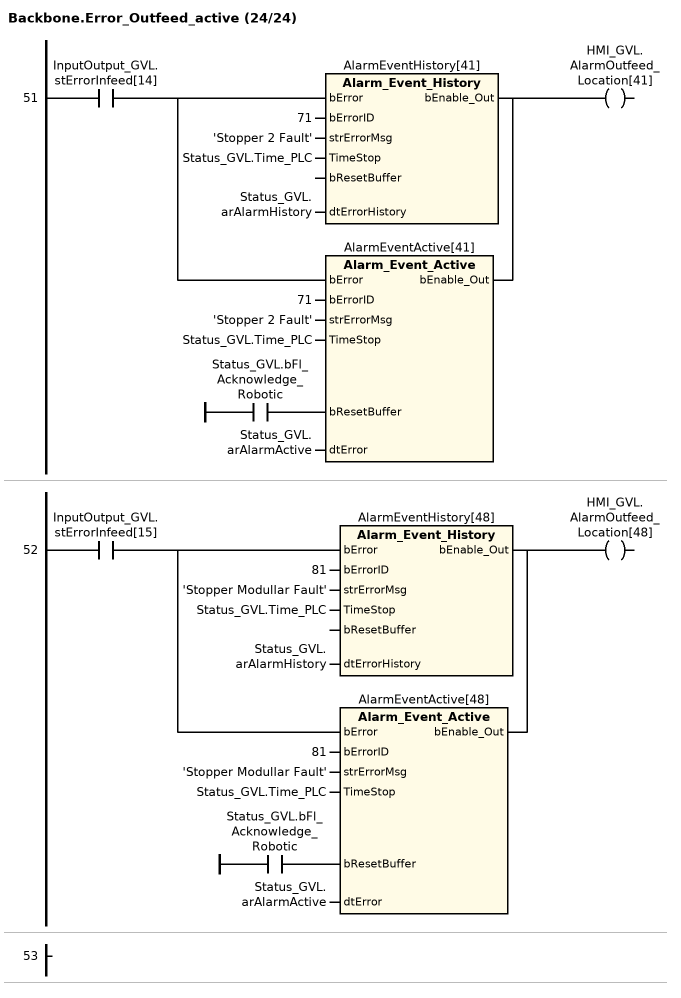
// NETWORK 51
AlarmEventHistory[41](
    bError := InputOutput_GVL.stErrorInfeed[14],
    bErrorID := 71,
    strErrorMsg := 'Stopper 2 Fault',
    TimeStop := Status_GVL.Time_PLC,
    dtErrorHistory := Status_GVL.arAlarmHistory); // Alarm_Event_History
AlarmEventActive[41](
    bError := InputOutput_GVL.stErrorInfeed[14],
    bErrorID := 71,
    strErrorMsg := 'Stopper 2 Fault',
    TimeStop := Status_GVL.Time_PLC,
    bResetBuffer := Status_GVL.bFl_Acknowledge_Robotic,
    dtError := Status_GVL.arAlarmActive); // Alarm_Event_Active
HMI_GVL.AlarmOutfeed_Location[41] := AlarmEventHistory[41].bEnable_Out OR AlarmEventActive[41].bEnable_Out;

// NETWORK 52
AlarmEventHistory[48](
    bError := InputOutput_GVL.stErrorInfeed[15],
    bErrorID := 81,
    strErrorMsg := 'Stopper Modullar Fault',
    TimeStop := Status_GVL.Time_PLC,
    dtErrorHistory := Status_GVL.arAlarmHistory); // Alarm_Event_History
AlarmEventActive[48](
    bError := InputOutput_GVL.stErrorInfeed[15],
    bErrorID := 81,
    strErrorMsg := 'Stopper Modullar Fault',
    TimeStop := Status_GVL.Time_PLC,
    bResetBuffer := Status_GVL.bFl_Acknowledge_Robotic,
    dtError := Status_GVL.arAlarmActive); // Alarm_Event_Active
HMI_GVL.AlarmOutfeed_Location[48] := AlarmEventHistory[48].bEnable_Out OR AlarmEventActive[48].bEnable_Out;

// NETWORK 53
END_ACTION

ACTION FGHS_DataCollect_active:
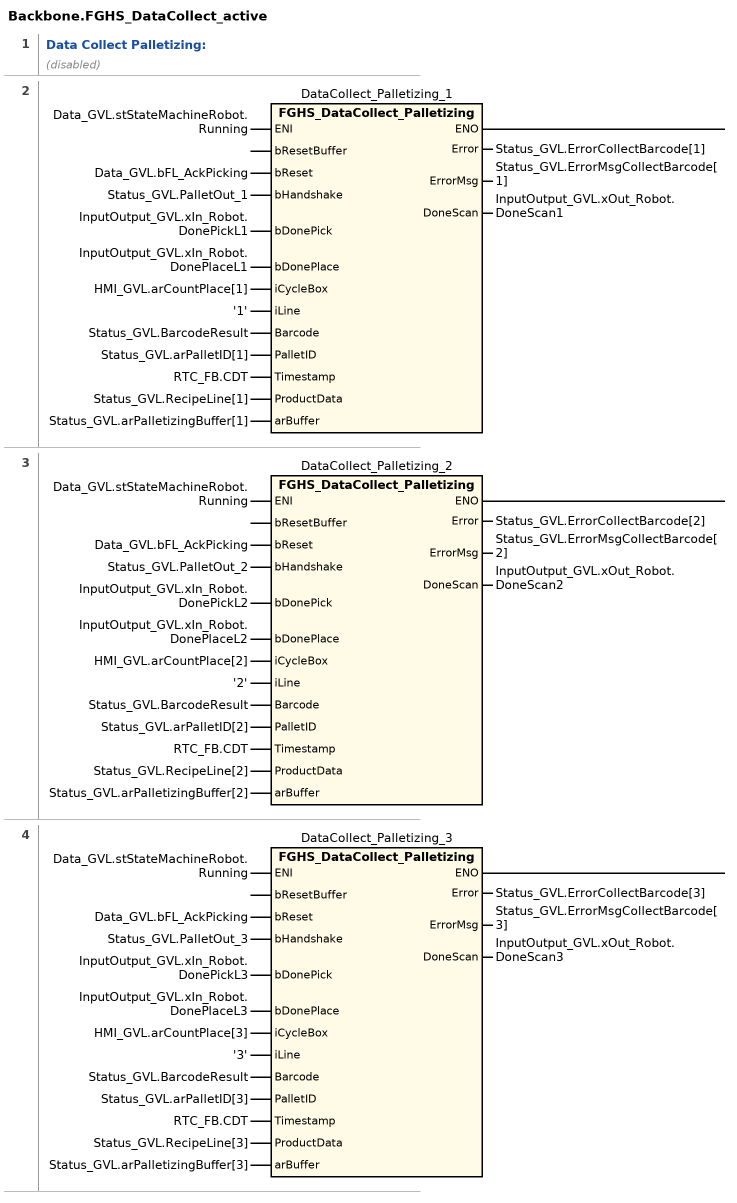
// NETWORK 1 (disabled)
// label: Data Collect Palletizing

// NETWORK 2
DataCollect_Palletizing_1(
    ENI := Data_GVL.stStateMachineRobot.Running,
    bReset := Data_GVL.bFL_AckPicking,
    bHandshake := Status_GVL.PalletOut_1,
    bDonePick := InputOutput_GVL.xIn_Robot.DonePickL1,
    bDonePlace := InputOutput_GVL.xIn_Robot.DonePlaceL1,
    iCycleBox := HMI_GVL.arCountPlace[1],
    iLine := '1',
    Barcode := Status_GVL.BarcodeResult,
    PalletID := Status_GVL.arPalletID[1],
    Timestamp := RTC_FB.CDT,
    ProductData := Status_GVL.RecipeLine[1],
    arBuffer := Status_GVL.arPalletizingBuffer[1],
    Error => Status_GVL.ErrorCollectBarcode[1],
    ErrorMsg => Status_GVL.ErrorMsgCollectBarcode[1],
    DoneScan => InputOutput_GVL.xOut_Robot.DoneScan1); // FGHS_DataCollect_Palletizing

// NETWORK 3
DataCollect_Palletizing_2(
    ENI := Data_GVL.stStateMachineRobot.Running,
    bReset := Data_GVL.bFL_AckPicking,
    bHandshake := Status_GVL.PalletOut_2,
    bDonePick := InputOutput_GVL.xIn_Robot.DonePickL2,
    bDonePlace := InputOutput_GVL.xIn_Robot.DonePlaceL2,
    iCycleBox := HMI_GVL.arCountPlace[2],
    iLine := '2',
    Barcode := Status_GVL.BarcodeResult,
    PalletID := Status_GVL.arPalletID[2],
    Timestamp := RTC_FB.CDT,
    ProductData := Status_GVL.RecipeLine[2],
    arBuffer := Status_GVL.arPalletizingBuffer[2],
    Error => Status_GVL.ErrorCollectBarcode[2],
    ErrorMsg => Status_GVL.ErrorMsgCollectBarcode[2],
    DoneScan => InputOutput_GVL.xOut_Robot.DoneScan2); // FGHS_DataCollect_Palletizing

// NETWORK 4
DataCollect_Palletizing_3(
    ENI := Data_GVL.stStateMachineRobot.Running,
    bReset := Data_GVL.bFL_AckPicking,
    bHandshake := Status_GVL.PalletOut_3,
    bDonePick := InputOutput_GVL.xIn_Robot.DonePickL3,
    bDonePlace := InputOutput_GVL.xIn_Robot.DonePlaceL3,
    iCycleBox := HMI_GVL.arCountPlace[3],
    iLine := '3',
    Barcode := Status_GVL.BarcodeResult,
    PalletID := Status_GVL.arPalletID[3],
    Timestamp := RTC_FB.CDT,
    ProductData := Status_GVL.RecipeLine[3],
    arBuffer := Status_GVL.arPalletizingBuffer[3],
    Error => Status_GVL.ErrorCollectBarcode[3],
    ErrorMsg => Status_GVL.ErrorMsgCollectBarcode[3],
    DoneScan => InputOutput_GVL.xOut_Robot.DoneScan3); // FGHS_DataCollect_Palletizing

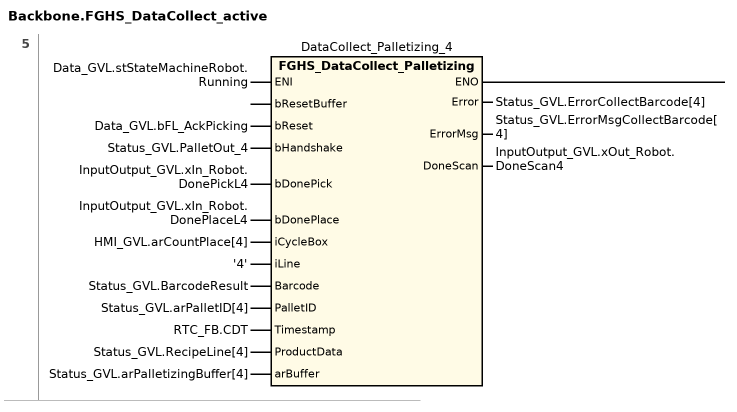
// NETWORK 5
DataCollect_Palletizing_4(
    ENI := Data_GVL.stStateMachineRobot.Running,
    bReset := Data_GVL.bFL_AckPicking,
    bHandshake := Status_GVL.PalletOut_4,
    bDonePick := InputOutput_GVL.xIn_Robot.DonePickL4,
    bDonePlace := InputOutput_GVL.xIn_Robot.DonePlaceL4,
    iCycleBox := HMI_GVL.arCountPlace[4],
    iLine := '4',
    Barcode := Status_GVL.BarcodeResult,
    PalletID := Status_GVL.arPalletID[4],
    Timestamp := RTC_FB.CDT,
    ProductData := Status_GVL.RecipeLine[4],
    arBuffer := Status_GVL.arPalletizingBuffer[4],
    Error => Status_GVL.ErrorCollectBarcode[4],
    ErrorMsg => Status_GVL.ErrorMsgCollectBarcode[4],
    DoneScan => InputOutput_GVL.xOut_Robot.DoneScan4); // FGHS_DataCollect_Palletizing
END_ACTION

ACTION FGHS_DataTraffict_active:
(* ============= Barcode Product ================= *)
//Line 1
	IF HMI_GVL.arCountReal[1] <> CheckCounter[1] THEN
		FOR Index[1] := 1 TO 60 BY 1 DO
		Status_GVL.arBarcodePallet[1,Index[1]]			:= Status_GVL.arPalletizingBuffer[1].BarcodeProduct[Index[1]];
		Status_GVL.arBarcodePalletTime[1,Index[1]]		:= Status_GVL.arPalletizingBuffer[1].BarcodeProductTime[Index[1]];
		Status_GVL.arDataPallet1[Index[1]].BarcodePallet	:= Status_GVL.arBarcodePallet[1,Index[1]];
		Status_GVL.arDataPallet1[Index[1]].BarcodePalletTime:= Status_GVL.arBarcodePalletTime[1,Index[1]]; 
		END_FOR
		CheckCounter[1]	:= HMI_GVL.arCountReal[1];
	END_IF
	
//Line 2
	IF HMI_GVL.arCountReal[2] <> CheckCounter[2] THEN
		FOR Index[2] := 1 TO 60 BY 1 DO
		Status_GVL.arBarcodePallet[2,Index[2]]			:= Status_GVL.arPalletizingBuffer[2].BarcodeProduct[Index[2]];
		Status_GVL.arBarcodePalletTime[2,Index[2]]		:= Status_GVL.arPalletizingBuffer[2].BarcodeProductTime[Index[2]];
		Status_GVL.arDataPallet2[Index[2]].BarcodePallet	:= Status_GVL.arBarcodePallet[2,Index[2]];
		Status_GVL.arDataPallet2[Index[2]].BarcodePalletTime:= Status_GVL.arBarcodePalletTime[2,Index[2]]; 
		END_FOR
		CheckCounter[2]	:= HMI_GVL.arCountReal[2];
	END_IF
	
//Line 3
	IF HMI_GVL.arCountReal[3] <> CheckCounter[3] THEN
		FOR Index[3] := 1 TO 60 BY 1 DO
		Status_GVL.arBarcodePallet[3,Index[3]]			:= Status_GVL.arPalletizingBuffer[3].BarcodeProduct[Index[3]];
		Status_GVL.arBarcodePalletTime[3,Index[3]]		:= Status_GVL.arPalletizingBuffer[3].BarcodeProductTime[Index[3]];
		Status_GVL.arDataPallet3[Index[3]].BarcodePallet	:= Status_GVL.arBarcodePallet[3,Index[3]];
		Status_GVL.arDataPallet3[Index[3]].BarcodePalletTime:= Status_GVL.arBarcodePalletTime[3,Index[3]]; 
		END_FOR
		CheckCounter[3]	:= HMI_GVL.arCountReal[3];
	END_IF
	
//Line 4
	IF HMI_GVL.arCountReal[4] <> CheckCounter[4] THEN
		FOR Index[4] := 1 TO 60 BY 1 DO
		Status_GVL.arBarcodePallet[4,Index[4]]			:= Status_GVL.arPalletizingBuffer[4].BarcodeProduct[Index[4]];
		Status_GVL.arBarcodePalletTime[4,Index[4]]		:= Status_GVL.arPalletizingBuffer[4].BarcodeProductTime[Index[4]];
		Status_GVL.arDataPallet4[Index[4]].BarcodePallet	:= Status_GVL.arBarcodePallet[4,Index[4]];
		Status_GVL.arDataPallet4[Index[4]].BarcodePalletTime:= Status_GVL.arBarcodePalletTime[4,Index[4]]; 
		END_FOR
		CheckCounter[4]	:= HMI_GVL.arCountReal[4];
	END_IF
	
	
(* ============= Link Up ================= *)
Status_GVl.arPallet_LinkUp[1]	:= Status_GVL.RecipeLine[1].LinkUpSource;
Status_GVl.arPallet_LinkUp[2]	:= Status_GVL.RecipeLine[2].LinkUpSource;
Status_GVl.arPallet_LinkUp[3]	:= Status_GVL.RecipeLine[3].LinkUpSource;
Status_GVl.arPallet_LinkUp[4]	:= Status_GVL.RecipeLine[4].LinkUpSource;


(* ============= EAN Variant ================= *)
Status_GVL.arCurrent_EAN[1]		:= Status_GVL.RecipeLine[1].EANVariant;
Status_GVL.arCurrent_EAN[2]		:= Status_GVL.RecipeLine[2].EANVariant;
Status_GVL.arCurrent_EAN[3]		:= Status_GVL.RecipeLine[3].EANVariant;
Status_GVL.arCurrent_EAN[4]		:= Status_GVL.RecipeLine[4].EANVariant;

(* ============= Code Variant ================= *)
Status_GVL.arCurrent_CodeVariant[1]		:= Status_GVL.RecipeLine[1].CodeVariant;
Status_GVL.arCurrent_CodeVariant[2]		:= Status_GVL.RecipeLine[2].CodeVariant;
Status_GVL.arCurrent_CodeVariant[3]		:= Status_GVL.RecipeLine[3].CodeVariant;
Status_GVL.arCurrent_CodeVariant[4]		:= Status_GVL.RecipeLine[4].CodeVariant;

(* ============= Interlock Infeed ================= *)
Status_GVL.ModullarInfeedBusy	:= InputOutput_GVL.Digital_Output[45];
END_ACTION

ACTION Indicator_active:
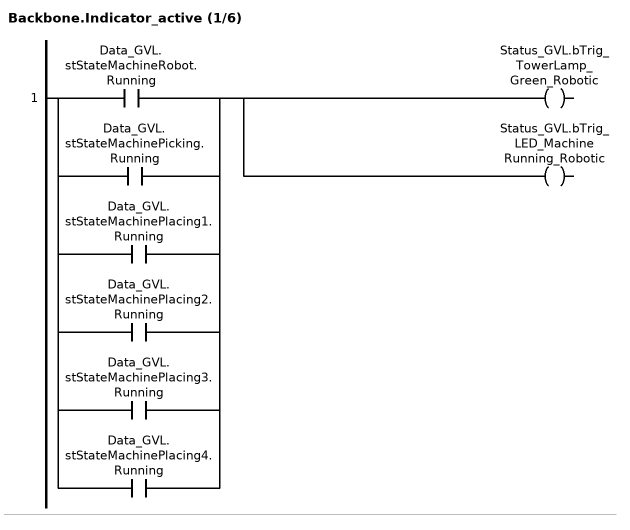
// NETWORK 1
_w1 := Data_GVL.stStateMachineRobot.Running OR Data_GVL.stStateMachinePicking.Running OR Data_GVL.stStateMachinePlacing1.Running OR Data_GVL.stStateMachinePlacing2.Running OR Data_GVL.stStateMachinePlacing3.Running OR Data_GVL.stStateMachinePlacing4.Running;
Status_GVL.bTrig_TowerLamp_Green_Robotic := _w1;
Status_GVL.bTrig_LED_MachineRunning_Robotic := _w1;

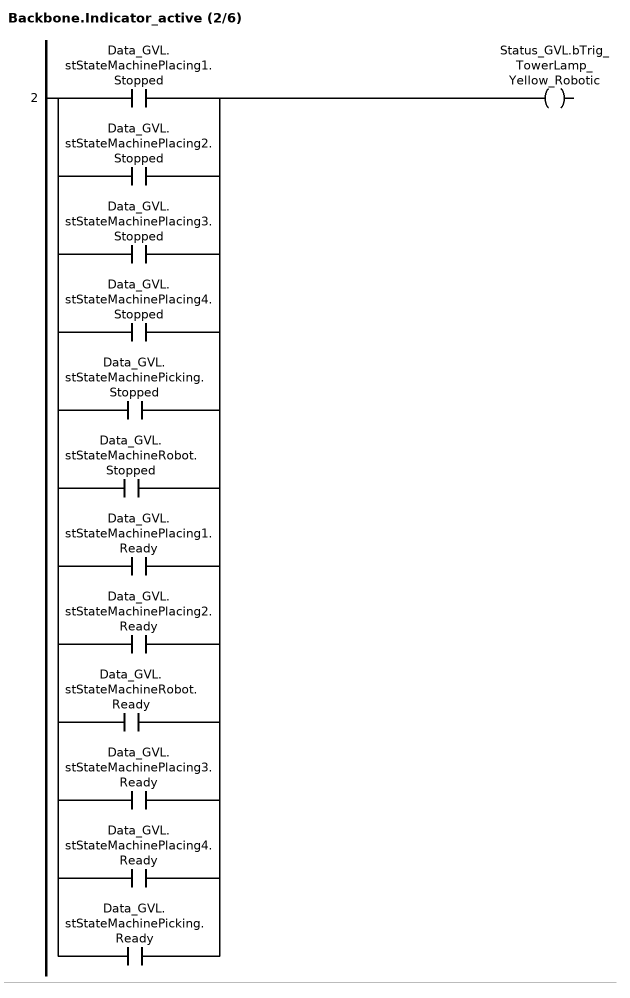
// NETWORK 2
Status_GVL.bTrig_TowerLamp_Yellow_Robotic := Data_GVL.stStateMachinePlacing1.Stopped OR Data_GVL.stStateMachinePlacing2.Stopped OR Data_GVL.stStateMachinePlacing3.Stopped OR Data_GVL.stStateMachinePlacing4.Stopped OR Data_GVL.stStateMachinePicking.Stopped OR Data_GVL.stStateMachineRobot.Stopped OR Data_GVL.stStateMachinePlacing1.Ready OR Data_GVL.stStateMachinePlacing2.Ready OR Data_GVL.stStateMachineRobot.Ready OR Data_GVL.stStateMachinePlacing3.Ready OR Data_GVL.stStateMachinePlacing4.Ready OR Data_GVL.stStateMachinePicking.Ready;

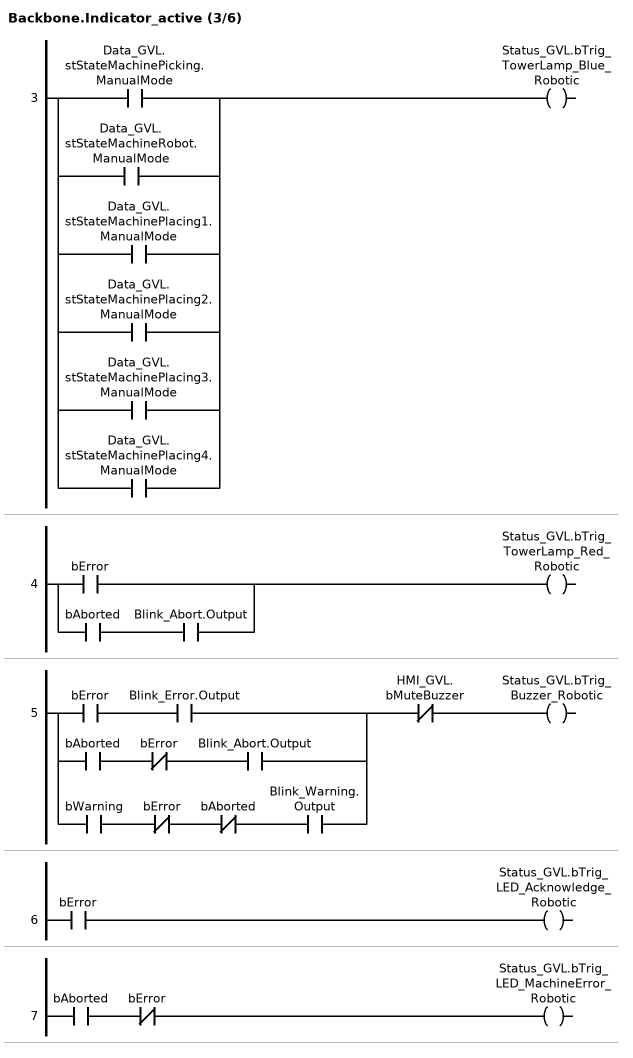
// NETWORK 3
Status_GVL.bTrig_TowerLamp_Blue_Robotic := Data_GVL.stStateMachinePicking.ManualMode OR Data_GVL.stStateMachineRobot.ManualMode OR Data_GVL.stStateMachinePlacing1.ManualMode OR Data_GVL.stStateMachinePlacing2.ManualMode OR Data_GVL.stStateMachinePlacing3.ManualMode OR Data_GVL.stStateMachinePlacing4.ManualMode;

// NETWORK 4
Status_GVL.bTrig_TowerLamp_Red_Robotic := bError OR bAborted AND Blink_Abort.Output;

// NETWORK 5
Status_GVL.bTrig_Buzzer_Robotic := (bError AND Blink_Error.Output OR bAborted AND NOT bError AND Blink_Abort.Output OR bWarning AND NOT bError AND NOT bAborted AND Blink_Warning.Output) AND NOT HMI_GVL.bMuteBuzzer;

// NETWORK 6
Status_GVL.bTrig_LED_Acknowledge_Robotic := bError;

// NETWORK 7
Status_GVL.bTrig_LED_MachineError_Robotic := bAborted AND NOT bError;

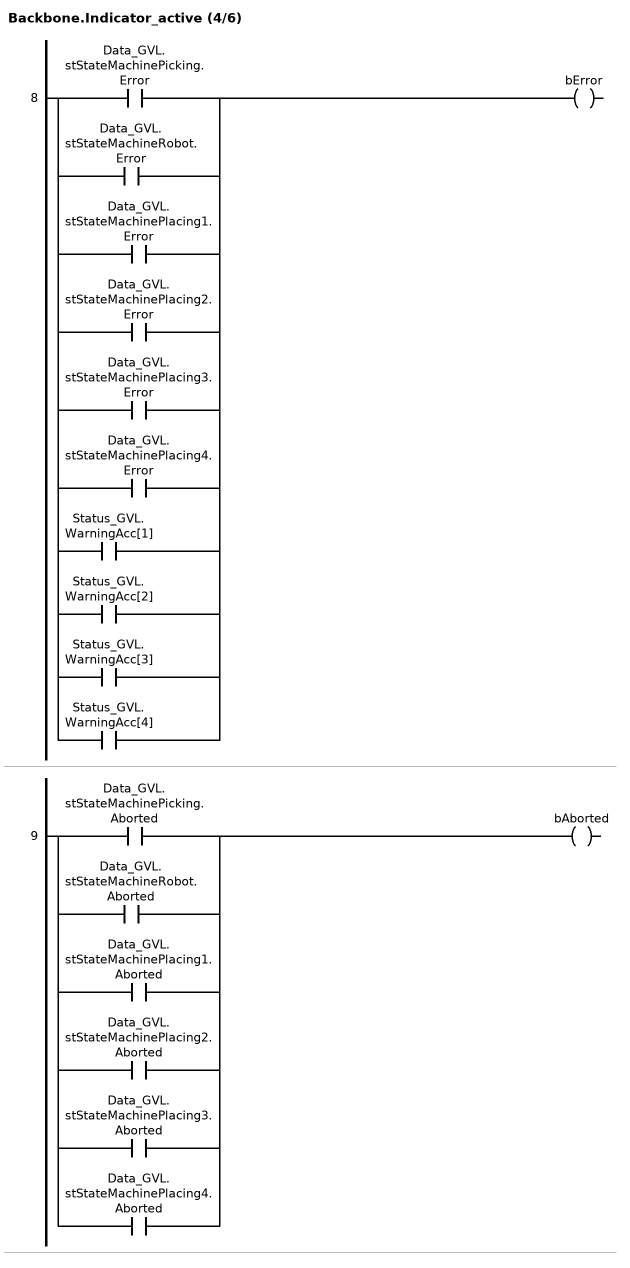
// NETWORK 8
bError := Data_GVL.stStateMachinePicking.Error OR Data_GVL.stStateMachineRobot.Error OR Data_GVL.stStateMachinePlacing1.Error OR Data_GVL.stStateMachinePlacing2.Error OR Data_GVL.stStateMachinePlacing3.Error OR Data_GVL.stStateMachinePlacing4.Error OR Status_GVL.WarningAcc[1] OR Status_GVL.WarningAcc[2] OR Status_GVL.WarningAcc[3] OR Status_GVL.WarningAcc[4];

// NETWORK 9
bAborted := Data_GVL.stStateMachinePicking.Aborted OR Data_GVL.stStateMachineRobot.Aborted OR Data_GVL.stStateMachinePlacing1.Aborted OR Data_GVL.stStateMachinePlacing2.Aborted OR Data_GVL.stStateMachinePlacing3.Aborted OR Data_GVL.stStateMachinePlacing4.Aborted;

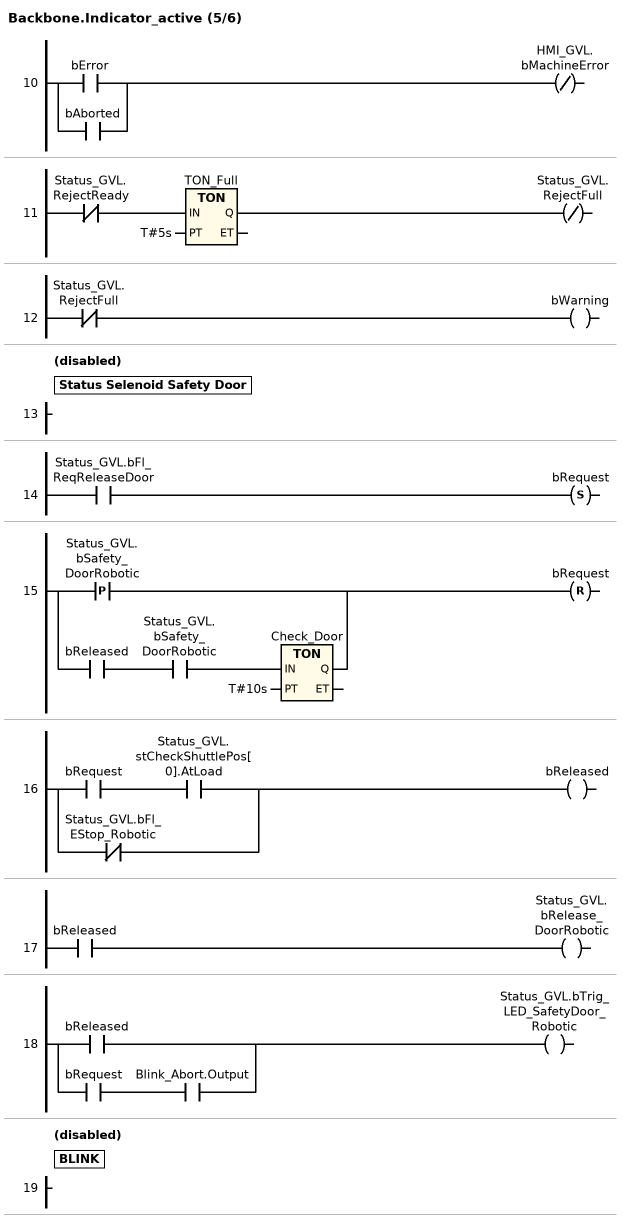
// NETWORK 10
HMI_GVL.bMachineError := NOT (bError OR bAborted);

// NETWORK 11
TON_Full(IN := NOT Status_GVL.RejectReady, PT := T#5s); // TON
Status_GVL.RejectFull := NOT TON_Full.Q;

// NETWORK 12
bWarning := NOT Status_GVL.RejectFull;

// NETWORK 13 (disabled)
// label: Status Selenoid Safety Door

// NETWORK 14
bRequest S= Status_GVL.bFl_ReqReleaseDoor;

// NETWORK 15
_rt1(CLK := Status_GVL.bSafety_DoorRobotic);
Check_Door(IN := bReleased AND Status_GVL.bSafety_DoorRobotic, PT := T#10s); // TON
bRequest R= _rt1.Q OR Check_Door.Q;

// NETWORK 16
bReleased := bRequest AND Status_GVL.stCheckShuttlePos[0].AtLoad OR NOT Status_GVL.bFl_EStop_Robotic;

// NETWORK 17
Status_GVL.bRelease_DoorRobotic := bReleased;

// NETWORK 18
Status_GVL.bTrig_LED_SafetyDoor_Robotic := bReleased OR bRequest AND Blink_Abort.Output;

// NETWORK 19 (disabled)
// label: BLINK

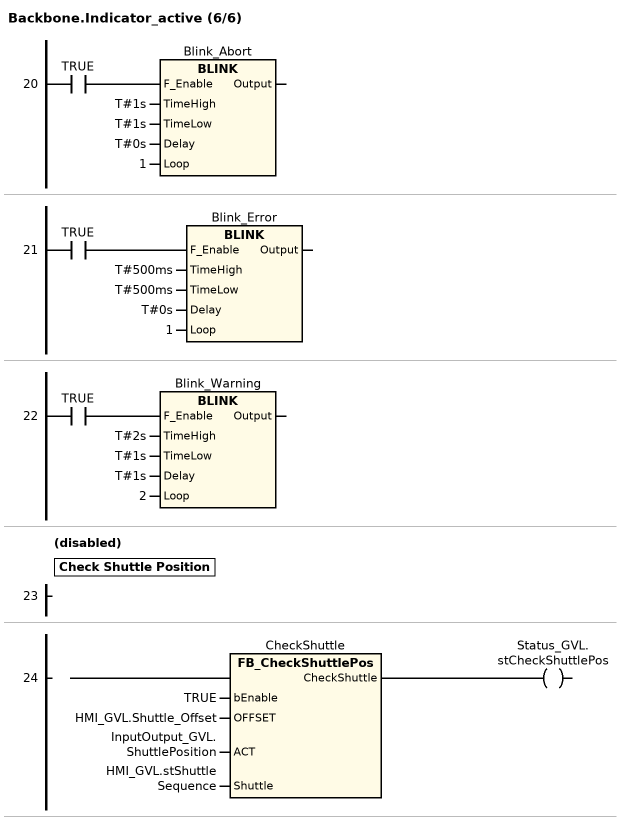
// NETWORK 20
Blink_Abort(F_Enable := TRUE, TimeHigh := T#1s, TimeLow := T#1s, Delay := T#0s, Loop := 1); // BLINK

// NETWORK 21
Blink_Error(F_Enable := TRUE, TimeHigh := T#500ms, TimeLow := T#500ms, Delay := T#0s, Loop := 1); // BLINK

// NETWORK 22
Blink_Warning(F_Enable := TRUE, TimeHigh := T#2s, TimeLow := T#1s, Delay := T#1s, Loop := 2); // BLINK

// NETWORK 23 (disabled)
// label: Check Shuttle Position

// NETWORK 24
CheckShuttle(
    bEnable := TRUE,
    OFFSET := HMI_GVL.Shuttle_Offset,
    ACT := InputOutput_GVL.ShuttlePosition,
    Shuttle := HMI_GVL.stShuttleSequence); // FB_CheckShuttlePos
Status_GVL.stCheckShuttlePos := CheckShuttle.CheckShuttle;
END_ACTION

ACTION OEE_active:
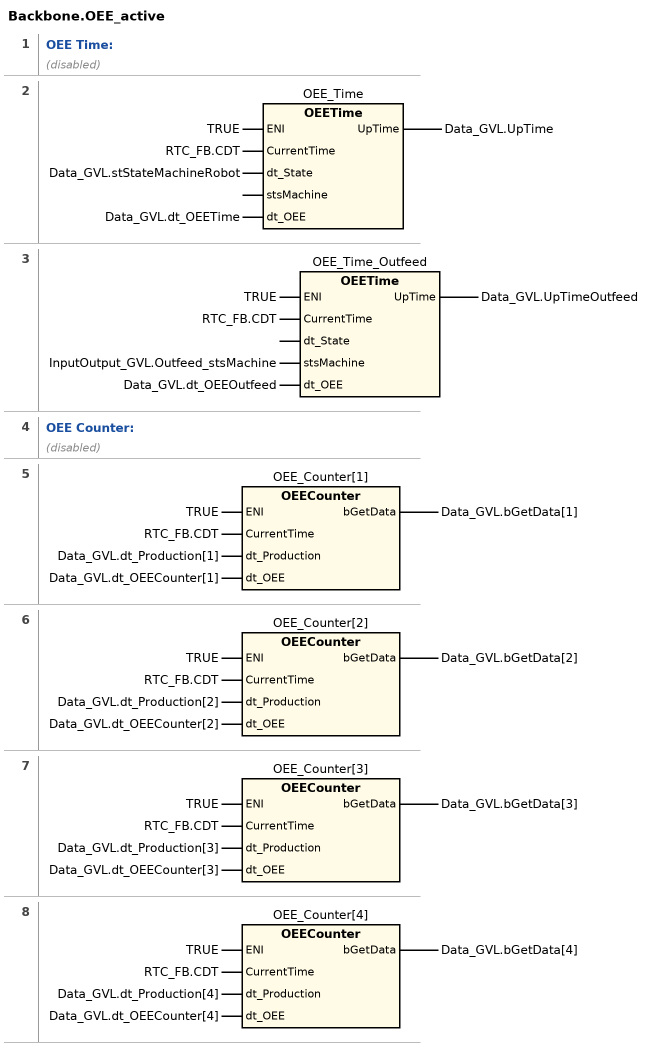
// NETWORK 1 (disabled)
// label: OEE Time

// NETWORK 2
OEE_Time(
    ENI := TRUE,
    CurrentTime := RTC_FB.CDT,
    dt_State := Data_GVL.stStateMachineRobot,
    dt_OEE := Data_GVL.dt_OEETime); // OEETime
Data_GVL.UpTime := OEE_Time.UpTime;

// NETWORK 3
OEE_Time_Outfeed(
    ENI := TRUE,
    CurrentTime := RTC_FB.CDT,
    stsMachine := InputOutput_GVL.Outfeed_stsMachine,
    dt_OEE := Data_GVL.dt_OEEOutfeed); // OEETime
Data_GVL.UpTimeOutfeed := OEE_Time_Outfeed.UpTime;

// NETWORK 4 (disabled)
// label: OEE Counter

// NETWORK 5
OEE_Counter[1](
    ENI := TRUE,
    CurrentTime := RTC_FB.CDT,
    dt_Production := Data_GVL.dt_Production[1],
    dt_OEE := Data_GVL.dt_OEECounter[1]); // OEECounter
Data_GVL.bGetData[1] := OEE_Counter[1].bGetData;

// NETWORK 6
OEE_Counter[2](
    ENI := TRUE,
    CurrentTime := RTC_FB.CDT,
    dt_Production := Data_GVL.dt_Production[2],
    dt_OEE := Data_GVL.dt_OEECounter[2]); // OEECounter
Data_GVL.bGetData[2] := OEE_Counter[2].bGetData;

// NETWORK 7
OEE_Counter[3](
    ENI := TRUE,
    CurrentTime := RTC_FB.CDT,
    dt_Production := Data_GVL.dt_Production[3],
    dt_OEE := Data_GVL.dt_OEECounter[3]); // OEECounter
Data_GVL.bGetData[3] := OEE_Counter[3].bGetData;

// NETWORK 8
OEE_Counter[4](
    ENI := TRUE,
    CurrentTime := RTC_FB.CDT,
    dt_Production := Data_GVL.dt_Production[4],
    dt_OEE := Data_GVL.dt_OEECounter[4]); // OEECounter
Data_GVL.bGetData[4] := OEE_Counter[4].bGetData;
END_ACTION

ACTION Parameter_Outfeed_active:
//Safety Outfeed
InputOutput_GVL.TestMode[99]	:= NOT Status_GVL.bFl_EStop_Robotic OR NOT Status_GVL.bSafety_DoorRobotic OR Backbone.bRequest;

//Mute Buzzer
InputOutput_GVL.TestMode[98]	:= HMI_GVL.bMuteBuzzer;

//Disable Overflow
InputOutput_GVL.TestMode[97]	:= HMI_GVL.Disable_Overflow;

//Lock Modullar to Keep Running
InputOutput_GVL.TestMode[96]	:= HMI_GVL.LockModullarToRun;

//Ack Button Outfeed
InputOutput_GVL.TestMode[95]	:= Status_GVL.bFl_Acknowledge_Robotic;

//Reset Button Outfeed
InputOutput_GVL.TestMode[94]	:= Status_GVL.bFl_ResetButton_Robotic;

//Status Running Picking
InputOutput_GVL.TestMode[93]	:= Data_GVL.stStateMachinePicking.Running;

//Bypass Wrapper
InputOutput_GVL.TestMode[92]	:= HMI_GVL.BypassWrapper;

//Bypass Wrapper Existing
InputOutput_GVL.TestMode[91]	:= HMI_GVL.BypassWrapperExisting;

(*================= Control Button ============================*) 
InputOutput_GVL.ControlButton[1]					:= HMI_GVL.bStartButtonOutfeed;
InputOutput_GVL.ControlButton[2]					:= HMI_GVL.bStopButtonOutfeed;
InputOutput_GVL.ControlButton[3]					:= HMI_GVL.bResetButtonOutfeed;
InputOutput_GVL.ControlButton[4]					:= HMI_GVL.bTestModeEnableOutfeed;
InputOutput_GVL.ControlButton[5]					:= HMI_GVL.bAcknowledgeButtonOutfeed;

InputOutput_GVL.ControlButton[6]					:= HMI_GVL.bStartButtonShuttle;
InputOutput_GVL.ControlButton[7]					:= HMI_GVL.bStopButtonShuttle;
InputOutput_GVL.ControlButton[8]					:= HMI_GVL.bResetButtonShuttle;
InputOutput_GVL.ControlButton[9]					:= HMI_GVL.bTestModeEnableShuttle;
InputOutput_GVL.ControlButton[10]					:= HMI_GVL.bAcknowledgeButtonShuttle;

InputOutput_GVL.ControlButton[11]					:= HMI_GVL.bStartButtonDispenser;
InputOutput_GVL.ControlButton[12]					:= HMI_GVL.bStopButtonDispenser;
InputOutput_GVL.ControlButton[13]					:= HMI_GVL.bResetButtonDispenser;
InputOutput_GVL.ControlButton[14]					:= HMI_GVL.bTestModeEnableDispenser;
InputOutput_GVL.ControlButton[15]					:= HMI_GVL.bAcknowledgeButtonDispenser;

InputOutput_GVL.ControlButton[16]					:= HMI_GVL.bStartButtonInfeed;
InputOutput_GVL.ControlButton[17]					:= HMI_GVL.bStopButtonInfeed;
InputOutput_GVL.ControlButton[18]					:= HMI_GVL.bResetButtonInfeed;
InputOutput_GVL.ControlButton[19]					:= HMI_GVL.bTestModeEnableInfeed;
InputOutput_GVL.ControlButton[20]					:= HMI_GVL.bAcknowledgeButtonInfeed;


(*================= Parameter Shuttle ============================*)
//Handshake Shuttle
InputOutput_GVL.RequestEmptyPallet[1]	:= Status_GVL.RequestEmptyPallet[1];
InputOutput_GVL.RequestEmptyPallet[2]	:= Status_GVL.RequestEmptyPallet[2];
InputOutput_GVL.RequestEmptyPallet[3]	:= Status_GVL.RequestEmptyPallet[3];
InputOutput_GVL.RequestEmptyPallet[4]	:= Status_GVL.RequestEmptyPallet[4];

InputOutput_GVL.RequestLoadPallet[1]	:= Status_GVL.RequestLoadPallet[1];
InputOutput_GVL.RequestLoadPallet[2]	:= Status_GVL.RequestLoadPallet[2];
InputOutput_GVL.RequestLoadPallet[3]	:= Status_GVL.RequestLoadPallet[3];
InputOutput_GVL.RequestLoadPallet[4]	:= Status_GVL.RequestLoadPallet[4];

Status_GVL.FB_RequestShuttle[1]			:= InputOutput_GVL.FB_RequestShuttle[1];
Status_GVL.FB_RequestShuttle[2]			:= InputOutput_GVL.FB_RequestShuttle[2];
Status_GVL.FB_RequestShuttle[3]			:= InputOutput_GVL.FB_RequestShuttle[3];
Status_GVL.FB_RequestShuttle[4]			:= InputOutput_GVL.FB_RequestShuttle[4];


//Shuttle Position
//InputOutput_GVL.TestMode[100] ==> Download Parameter Shuttle Position	
InputOutput_GVL.stShuttleSequence[0].PositionEmpty	:= HMI_GVL.stShuttleSequence[0].PositionEmpty;
InputOutput_GVL.stShuttleSequence[1].PositionEmpty	:= HMI_GVL.stShuttleSequence[1].PositionEmpty;
InputOutput_GVL.stShuttleSequence[2].PositionEmpty	:= HMI_GVL.stShuttleSequence[2].PositionEmpty;
InputOutput_GVL.stShuttleSequence[3].PositionEmpty	:= HMI_GVL.stShuttleSequence[3].PositionEmpty;
InputOutput_GVL.stShuttleSequence[4].PositionEmpty	:= HMI_GVL.stShuttleSequence[4].PositionEmpty;

InputOutput_GVL.stShuttleSequence[0].PositionLoaded	:= HMI_GVL.stShuttleSequence[0].PositionLoaded;
InputOutput_GVL.stShuttleSequence[1].PositionLoaded	:= HMI_GVL.stShuttleSequence[1].PositionLoaded;
InputOutput_GVL.stShuttleSequence[2].PositionLoaded	:= HMI_GVL.stShuttleSequence[2].PositionLoaded;
InputOutput_GVL.stShuttleSequence[3].PositionLoaded	:= HMI_GVL.stShuttleSequence[3].PositionLoaded;
InputOutput_GVL.stShuttleSequence[4].PositionLoaded	:= HMI_GVL.stShuttleSequence[4].PositionLoaded;

//Shuttle Speed
InputOutput_GVL.Shuttle_Speed[1]					:= HMI_GVL.Shuttle_JogSpeed;
InputOutput_GVL.Shuttle_Speed[2]					:= HMI_GVL.Shuttle_MinSpeed;
InputOutput_GVL.Shuttle_Speed[3]					:= HMI_GVL.Shuttle_MaxSpeed;
InputOutput_GVL.Shuttle_Offset						:= HMI_GVL.Shuttle_Offset;

//Counter Box at Placing
InputOutput_GVL.Counter[1]							:= HMI_GVL.arCountReal[1];
InputOutput_GVL.Counter[2]							:= HMI_GVL.arCountReal[2];
InputOutput_GVL.Counter[3]							:= HMI_GVL.arCountReal[3];
InputOutput_GVL.Counter[4]							:= HMI_GVL.arCountReal[4];


(*================= Parameter Timer ============================*)
//=====> Shuttle
InputOutput_GVL.TmrOutfeed[1]						:= HMI_GVL.Tmr_EmptyShuttle;
InputOutput_GVL.TmrOutfeed[2]						:= HMI_GVL.Tmr_LoadedShuttle;
InputOutput_GVL.TmrOutfeed[3]						:= HMI_GVL.Tmr_BrakeShuttle; 

//=====> Outfeed
InputOutput_GVL.TmrOutfeed[4]						:= HMI_GVL.Tmr_PalletBuffer2;
InputOutput_GVL.TmrOutfeed[5]						:= HMI_GVL.Tmr_PalletBuffer1;
InputOutput_GVL.TmrOutfeed[6]						:= HMI_GVL.Tmr_PalletOutfeed1;
InputOutput_GVL.TmrOutfeed[7]						:= HMI_GVL.Tmr_PalletOutfeed2;
InputOutput_GVL.TmrOutfeed[8]						:= HMI_GVL.Tmr_PalletOutfeed3;
InputOutput_GVL.TmrOutfeed[9]						:= HMI_GVL.Tmr_PalletOutfeed4;
InputOutput_GVL.TmrOutfeed[10]						:= HMI_GVL.Tmr_PalletOutfeed5;
InputOutput_GVL.TmrOutfeed[11]						:= HMI_GVL.Tmr_PalletRA;
InputOutput_GVL.TmrOutfeed[12]						:= HMI_GVL.TmrDelay_PalletRA;

//=====> Infeed
InputOutput_GVL.TmrOutfeed[13]						:= HMI_GVL.Tmr_Stopper1;
InputOutput_GVL.TmrOutfeed[14]						:= HMI_GVL.Tmr_Stopper2;
InputOutput_GVL.TmrOutfeed[15]						:= HMI_GVL.Tmr_StopGo;
InputOutput_GVL.TmrOutfeed[16]						:= HMI_GVL.Tmr_Infeed;
InputOutput_GVL.TmrOutfeed[17]						:= HMI_GVL.Tmr_Buffer1;
InputOutput_GVL.TmrOutfeed[18]						:= HMI_GVL.Tmr_Buffer2;
InputOutput_GVL.TmrOutfeed[19]						:= HMI_GVL.Tmr_ModullarOn;
InputOutput_GVL.TmrOutfeed[20]						:= HMI_GVL.Tmr_ModullarOff;

//=====> Dispenser
InputOutput_GVL.TmrOutfeed[21]						:= HMI_GVL.Tmr_Dispenser;

(*================= SeqIndex ============================*)
//Shuttle Empty
CASE InputOutput_GVL.SeqIndexOutfeed[1] OF
	0:		HMI_GVL.CJ_ShuttleEmpty	:= 'Check Sensor';
	100:	HMI_GVL.CJ_ShuttleEmpty	:= 'Request to Dispenser';
	110:	HMI_GVL.CJ_ShuttleEmpty	:= 'Empty Pallet In';
	500:	HMI_GVL.CJ_ShuttleEmpty	:= 'Empty Pallet Ready';
	600:	HMI_GVL.CJ_ShuttleEmpty	:= 'Empty Pallet Out';
END_CASE

//Shuttle Load
CASE InputOutput_GVL.SeqIndexOutfeed[2] OF
	0:		HMI_GVL.CJ_ShuttleLoad	:= 'Check Sensor';
	100:	HMI_GVL.CJ_ShuttleLoad	:= 'Waiting to Pick Up Loaded Pallet';
	101:	HMI_GVL.CJ_ShuttleLoad	:= 'Unloading Pallet In';
	110:	HMI_GVL.CJ_ShuttleLoad	:= 'Loaded Pallet In';
	500:	HMI_GVL.CJ_ShuttleLoad	:= 'Loaded Pallet Ready';
	600:	HMI_GVL.CJ_ShuttleLoad	:= 'Loaded Pallet Out';
END_CASE


//Shuttle Management
CASE InputOutput_GVL.SeqIndexOutfeed[3] OF
	0:		HMI_GVL.CJ_ShuttleManagement	:= 'Standby';
	100:	HMI_GVL.CJ_ShuttleManagement	:= 'Move to Standby';
	
	1001:	HMI_GVL.CJ_ShuttleManagement	:= 'Move to Dispenser - Outfeed';
	1020:	HMI_GVL.CJ_ShuttleManagement	:= 'Shuttle at Dispenser - Outfeed';
	1030:	HMI_GVL.CJ_ShuttleManagement	:= 'Transfer Pallet at Dispenser - Outfeed';
	1100:	HMI_GVL.CJ_ShuttleManagement	:= 'Done Transfer Pallet at Dispenser - Outfeed';
	
	2001:	HMI_GVL.CJ_ShuttleManagement	:= 'Move to Unloading';
	2020:	HMI_GVL.CJ_ShuttleManagement	:= 'Request Load Pallet from Unloading';
	2030:	HMI_GVL.CJ_ShuttleManagement	:= 'Unloading Pallet In';
	2040:	HMI_GVL.CJ_ShuttleManagement	:= 'Check Request from Outfeed';
	2050:	HMI_GVL.CJ_ShuttleManagement	:= 'Transfer Load Pallet to Outfeed';
	2100:	HMI_GVL.CJ_ShuttleManagement	:= 'Done Unloading';
	
	3000:	HMI_GVL.CJ_ShuttleManagement	:= 'Waiting for Request Line';
	3001:	HMI_GVL.CJ_ShuttleManagement	:= 'Waiting for Request Line';
	3002:	HMI_GVL.CJ_ShuttleManagement	:= 'Waiting for Request Line';
	3003:	HMI_GVL.CJ_ShuttleManagement	:= 'Waiting for Request Line';
	3004:	HMI_GVL.CJ_ShuttleManagement	:= 'Waiting for Request Line';
	3011:	HMI_GVL.CJ_ShuttleManagement	:= 'Loaded Pallet Transfer From Line 1';
	3012:	HMI_GVL.CJ_ShuttleManagement	:= 'Loaded Pallet Transfer From Line 2';
	3013:	HMI_GVL.CJ_ShuttleManagement	:= 'Loaded Pallet Transfer From Line 3';
	3014:	HMI_GVL.CJ_ShuttleManagement	:= 'Loaded Pallet Transfer From Line 4';
	3041:	HMI_GVL.CJ_ShuttleManagement	:= 'Transfer Load Pallet from Line 1';
	3042:	HMI_GVL.CJ_ShuttleManagement	:= 'Transfer Load Pallet from Line 2';
	3043:	HMI_GVL.CJ_ShuttleManagement	:= 'Transfer Load Pallet from Line 3';
	3044:	HMI_GVL.CJ_ShuttleManagement	:= 'Transfer Load Pallet from Line 4';
	3051:	HMI_GVL.CJ_ShuttleManagement	:= 'Empty Pallet Transfer To Line 1';
	3052:	HMI_GVL.CJ_ShuttleManagement	:= 'Empty Pallet Transfer To Line 2';
	3053:	HMI_GVL.CJ_ShuttleManagement	:= 'Empty Pallet Transfer To Line 3';
	3054:	HMI_GVL.CJ_ShuttleManagement	:= 'Empty Pallet Transfer To Line 4';
	3091:	HMI_GVL.CJ_ShuttleManagement	:= 'Transfer Empty Pallet to Line 1';
	3092:	HMI_GVL.CJ_ShuttleManagement	:= 'Transfer Empty Pallet to Line 2';
	3093:	HMI_GVL.CJ_ShuttleManagement	:= 'Transfer Empty Pallet to Line 3';
	3094:	HMI_GVL.CJ_ShuttleManagement	:= 'Transfer Empty Pallet to Line 4';
	3100:	HMI_GVL.CJ_ShuttleManagement	:= 'Done Standby';
	
END_CASE

//Dispenser
CASE InputOutput_GVL.SeqIndexOutfeed[4] OF
	0:		HMI_GVL.CJ_Dispenser	:= 'Check Pallet';
	10:		HMI_GVL.CJ_Dispenser	:= 'Move Pneu Vertical to Middle';
	20:		HMI_GVL.CJ_Dispenser	:= 'Check Sensor Stack';
	50:		HMI_GVL.CJ_Dispenser	:= 'Pneu Horizontal Retract';
	100:	HMI_GVL.CJ_Dispenser	:= 'Move Pneu Vertical to Bottom';
	150:	HMI_GVL.CJ_Dispenser	:= 'Request Pallet';
	200:	HMI_GVL.CJ_Dispenser	:= 'Pallet In';
	500:	HMI_GVL.CJ_Dispenser	:= 'Check Stack Pallet';
	520:	HMI_GVL.CJ_Dispenser	:= 'Pneu Horizontal Retract';
	550:	HMI_GVL.CJ_Dispenser	:= 'Move Pneu Vertical to Middle';
	555:	HMI_GVL.CJ_Dispenser	:= 'Move Pneu Vertical to Middle';
	600:	HMI_GVL.CJ_Dispenser	:= 'Pneu Horizontal Advance';
	650:	HMI_GVL.CJ_Dispenser	:= 'Move Pneu Vertical to Top';
	700:	HMI_GVL.CJ_Dispenser	:= 'Transfer Pallet Out';
	750:	HMI_GVL.CJ_Dispenser	:= 'Move Pneu Vertical to Bottom';
	800:	HMI_GVL.CJ_Dispenser	:= 'Pneu Horizontal Retract';
	
END_CASE
END_ACTION

ACTION Recipe_active:
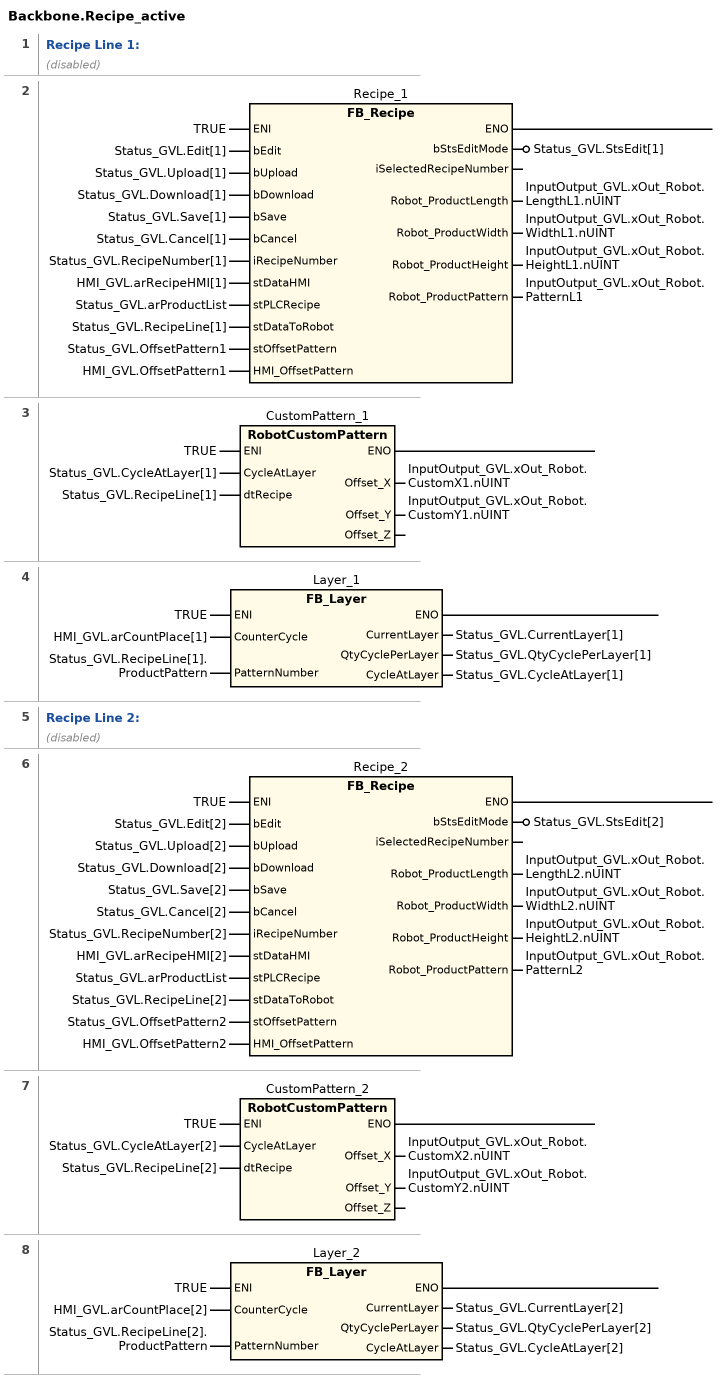
// NETWORK 1 (disabled)
// label: Recipe Line 1

// NETWORK 2
Recipe_1(
    ENI := TRUE,
    bEdit := Status_GVL.Edit[1],
    bUpload := Status_GVL.Upload[1],
    bDownload := Status_GVL.Download[1],
    bSave := Status_GVL.Save[1],
    bCancel := Status_GVL.Cancel[1],
    iRecipeNumber := Status_GVL.RecipeNumber[1],
    stDataHMI := HMI_GVL.arRecipeHMI[1],
    stPLCRecipe := Status_GVL.arProductList,
    stDataToRobot := Status_GVL.RecipeLine[1],
    stOffsetPattern := Status_GVL.OffsetPattern1,
    HMI_OffsetPattern := HMI_GVL.OffsetPattern1,
    Robot_ProductLength => InputOutput_GVL.xOut_Robot.LengthL1.nUINT,
    Robot_ProductWidth => InputOutput_GVL.xOut_Robot.WidthL1.nUINT,
    Robot_ProductHeight => InputOutput_GVL.xOut_Robot.HeightL1.nUINT,
    Robot_ProductPattern => InputOutput_GVL.xOut_Robot.PatternL1); // FB_Recipe
Status_GVL.StsEdit[1] := NOT Recipe_1.bStsEditMode;

// NETWORK 3
CustomPattern_1(
    ENI := TRUE,
    CycleAtLayer := Status_GVL.CycleAtLayer[1],
    dtRecipe := Status_GVL.RecipeLine[1],
    Offset_X => InputOutput_GVL.xOut_Robot.CustomX1.nUINT,
    Offset_Y => InputOutput_GVL.xOut_Robot.CustomY1.nUINT); // RobotCustomPattern

// NETWORK 4
Layer_1(
    ENI := TRUE,
    CounterCycle := HMI_GVL.arCountPlace[1],
    PatternNumber := Status_GVL.RecipeLine[1].ProductPattern,
    CurrentLayer => Status_GVL.CurrentLayer[1],
    QtyCyclePerLayer => Status_GVL.QtyCyclePerLayer[1],
    CycleAtLayer => Status_GVL.CycleAtLayer[1]); // FB_Layer

// NETWORK 5 (disabled)
// label: Recipe Line 2

// NETWORK 6
Recipe_2(
    ENI := TRUE,
    bEdit := Status_GVL.Edit[2],
    bUpload := Status_GVL.Upload[2],
    bDownload := Status_GVL.Download[2],
    bSave := Status_GVL.Save[2],
    bCancel := Status_GVL.Cancel[2],
    iRecipeNumber := Status_GVL.RecipeNumber[2],
    stDataHMI := HMI_GVL.arRecipeHMI[2],
    stPLCRecipe := Status_GVL.arProductList,
    stDataToRobot := Status_GVL.RecipeLine[2],
    stOffsetPattern := Status_GVL.OffsetPattern2,
    HMI_OffsetPattern := HMI_GVL.OffsetPattern2,
    Robot_ProductLength => InputOutput_GVL.xOut_Robot.LengthL2.nUINT,
    Robot_ProductWidth => InputOutput_GVL.xOut_Robot.WidthL2.nUINT,
    Robot_ProductHeight => InputOutput_GVL.xOut_Robot.HeightL2.nUINT,
    Robot_ProductPattern => InputOutput_GVL.xOut_Robot.PatternL2); // FB_Recipe
Status_GVL.StsEdit[2] := NOT Recipe_2.bStsEditMode;

// NETWORK 7
CustomPattern_2(
    ENI := TRUE,
    CycleAtLayer := Status_GVL.CycleAtLayer[2],
    dtRecipe := Status_GVL.RecipeLine[2],
    Offset_X => InputOutput_GVL.xOut_Robot.CustomX2.nUINT,
    Offset_Y => InputOutput_GVL.xOut_Robot.CustomY2.nUINT); // RobotCustomPattern

// NETWORK 8
Layer_2(
    ENI := TRUE,
    CounterCycle := HMI_GVL.arCountPlace[2],
    PatternNumber := Status_GVL.RecipeLine[2].ProductPattern,
    CurrentLayer => Status_GVL.CurrentLayer[2],
    QtyCyclePerLayer => Status_GVL.QtyCyclePerLayer[2],
    CycleAtLayer => Status_GVL.CycleAtLayer[2]); // FB_Layer

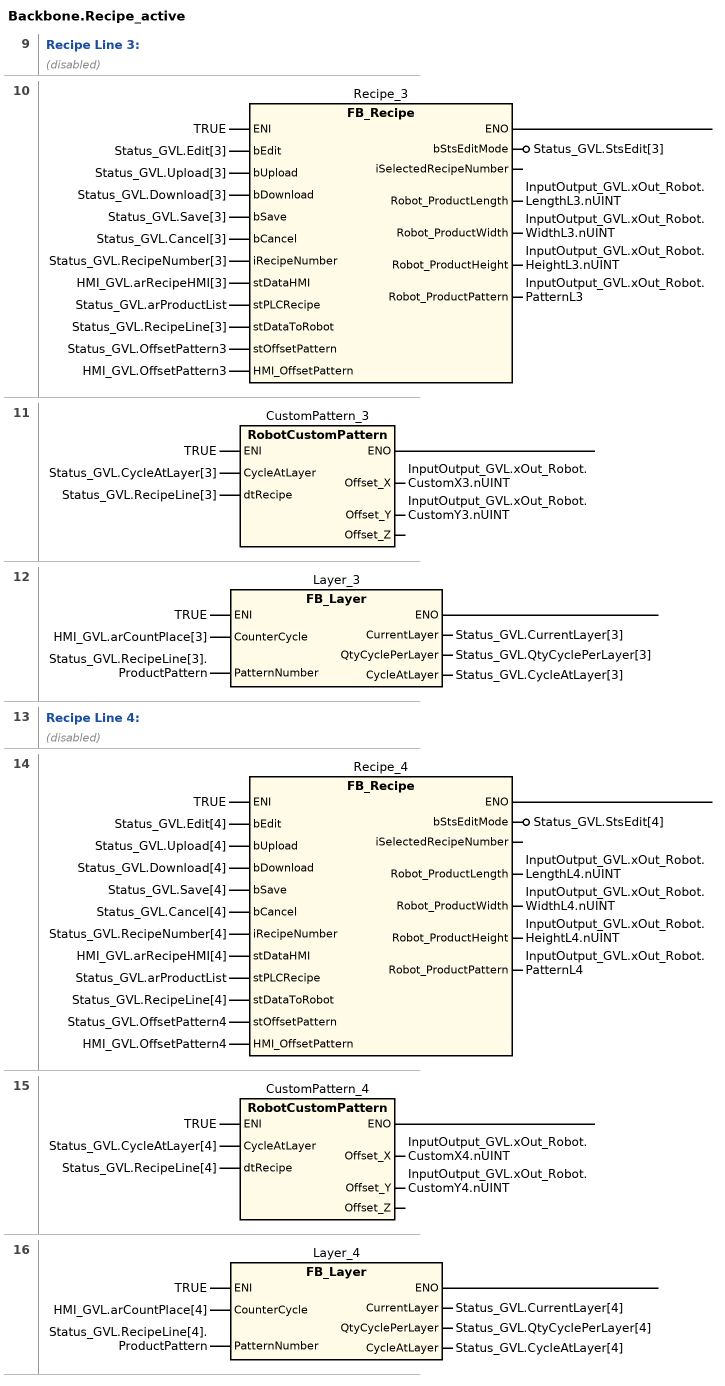
// NETWORK 9 (disabled)
// label: Recipe Line 3

// NETWORK 10
Recipe_3(
    ENI := TRUE,
    bEdit := Status_GVL.Edit[3],
    bUpload := Status_GVL.Upload[3],
    bDownload := Status_GVL.Download[3],
    bSave := Status_GVL.Save[3],
    bCancel := Status_GVL.Cancel[3],
    iRecipeNumber := Status_GVL.RecipeNumber[3],
    stDataHMI := HMI_GVL.arRecipeHMI[3],
    stPLCRecipe := Status_GVL.arProductList,
    stDataToRobot := Status_GVL.RecipeLine[3],
    stOffsetPattern := Status_GVL.OffsetPattern3,
    HMI_OffsetPattern := HMI_GVL.OffsetPattern3,
    Robot_ProductLength => InputOutput_GVL.xOut_Robot.LengthL3.nUINT,
    Robot_ProductWidth => InputOutput_GVL.xOut_Robot.WidthL3.nUINT,
    Robot_ProductHeight => InputOutput_GVL.xOut_Robot.HeightL3.nUINT,
    Robot_ProductPattern => InputOutput_GVL.xOut_Robot.PatternL3); // FB_Recipe
Status_GVL.StsEdit[3] := NOT Recipe_3.bStsEditMode;

// NETWORK 11
CustomPattern_3(
    ENI := TRUE,
    CycleAtLayer := Status_GVL.CycleAtLayer[3],
    dtRecipe := Status_GVL.RecipeLine[3],
    Offset_X => InputOutput_GVL.xOut_Robot.CustomX3.nUINT,
    Offset_Y => InputOutput_GVL.xOut_Robot.CustomY3.nUINT); // RobotCustomPattern

// NETWORK 12
Layer_3(
    ENI := TRUE,
    CounterCycle := HMI_GVL.arCountPlace[3],
    PatternNumber := Status_GVL.RecipeLine[3].ProductPattern,
    CurrentLayer => Status_GVL.CurrentLayer[3],
    QtyCyclePerLayer => Status_GVL.QtyCyclePerLayer[3],
    CycleAtLayer => Status_GVL.CycleAtLayer[3]); // FB_Layer

// NETWORK 13 (disabled)
// label: Recipe Line 4

// NETWORK 14
Recipe_4(
    ENI := TRUE,
    bEdit := Status_GVL.Edit[4],
    bUpload := Status_GVL.Upload[4],
    bDownload := Status_GVL.Download[4],
    bSave := Status_GVL.Save[4],
    bCancel := Status_GVL.Cancel[4],
    iRecipeNumber := Status_GVL.RecipeNumber[4],
    stDataHMI := HMI_GVL.arRecipeHMI[4],
    stPLCRecipe := Status_GVL.arProductList,
    stDataToRobot := Status_GVL.RecipeLine[4],
    stOffsetPattern := Status_GVL.OffsetPattern4,
    HMI_OffsetPattern := HMI_GVL.OffsetPattern4,
    Robot_ProductLength => InputOutput_GVL.xOut_Robot.LengthL4.nUINT,
    Robot_ProductWidth => InputOutput_GVL.xOut_Robot.WidthL4.nUINT,
    Robot_ProductHeight => InputOutput_GVL.xOut_Robot.HeightL4.nUINT,
    Robot_ProductPattern => InputOutput_GVL.xOut_Robot.PatternL4); // FB_Recipe
Status_GVL.StsEdit[4] := NOT Recipe_4.bStsEditMode;

// NETWORK 15
CustomPattern_4(
    ENI := TRUE,
    CycleAtLayer := Status_GVL.CycleAtLayer[4],
    dtRecipe := Status_GVL.RecipeLine[4],
    Offset_X => InputOutput_GVL.xOut_Robot.CustomX4.nUINT,
    Offset_Y => InputOutput_GVL.xOut_Robot.CustomY4.nUINT); // RobotCustomPattern

// NETWORK 16
Layer_4(
    ENI := TRUE,
    CounterCycle := HMI_GVL.arCountPlace[4],
    PatternNumber := Status_GVL.RecipeLine[4].ProductPattern,
    CurrentLayer => Status_GVL.CurrentLayer[4],
    QtyCyclePerLayer => Status_GVL.QtyCyclePerLayer[4],
    CycleAtLayer => Status_GVL.CycleAtLayer[4]); // FB_Layer

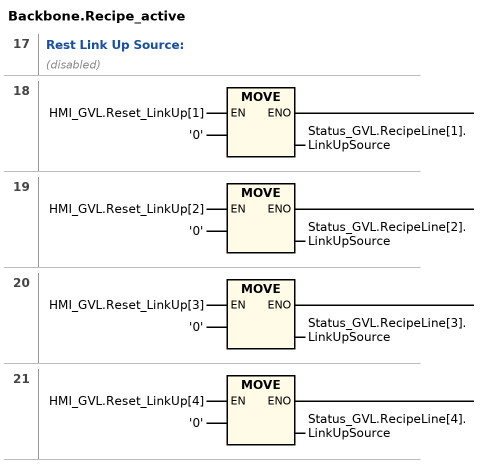
// NETWORK 17 (disabled)
// label: Rest Link Up Source

// NETWORK 18
IF HMI_GVL.Reset_LinkUp[1] THEN Status_GVL.RecipeLine[1].LinkUpSource := '0'; END_IF

// NETWORK 19
IF HMI_GVL.Reset_LinkUp[2] THEN Status_GVL.RecipeLine[2].LinkUpSource := '0'; END_IF

// NETWORK 20
IF HMI_GVL.Reset_LinkUp[3] THEN Status_GVL.RecipeLine[3].LinkUpSource := '0'; END_IF

// NETWORK 21
IF HMI_GVL.Reset_LinkUp[4] THEN Status_GVL.RecipeLine[4].LinkUpSource := '0'; END_IF
END_ACTION

ACTION RTC_Management_active:
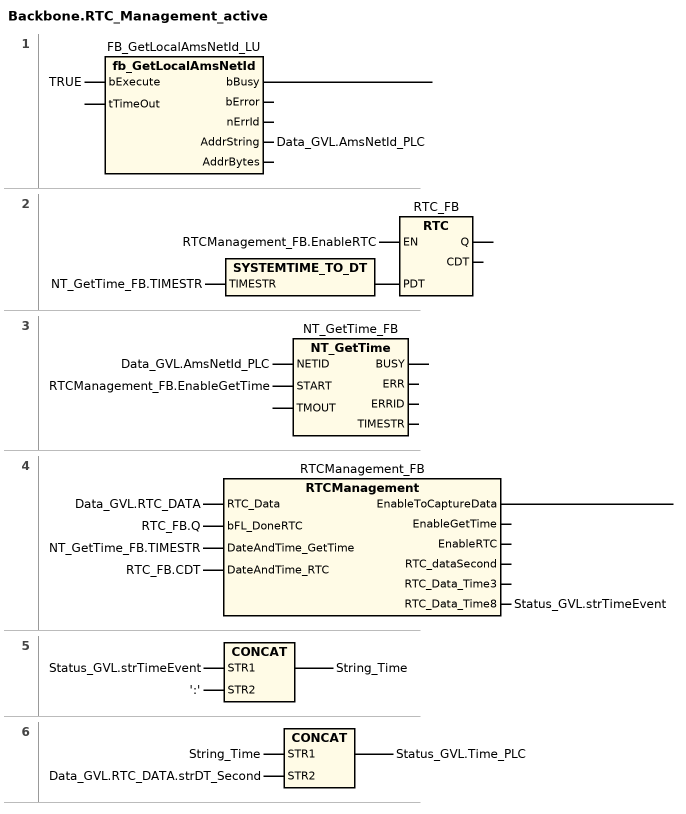
// NETWORK 1
FB_GetLocalAmsNetId_LU(bExecute := TRUE, AddrString => Data_GVL.AmsNetId_PLC); // fb_GetLocalAmsNetId

// NETWORK 2
RTC_FB(EN := RTCManagement_FB.EnableRTC, PDT := SYSTEMTIME_TO_DT(TIMESTR := NT_GetTime_FB.TIMESTR)); // RTC

// NETWORK 3
NT_GetTime_FB(NETID := Data_GVL.AmsNetId_PLC, START := RTCManagement_FB.EnableGetTime); // NT_GetTime

// NETWORK 4
RTCManagement_FB(
    RTC_Data := Data_GVL.RTC_DATA,
    bFL_DoneRTC := RTC_FB.Q,
    DateAndTime_GetTime := NT_GetTime_FB.TIMESTR,
    DateAndTime_RTC := RTC_FB.CDT,
    RTC_Data_Time8 => Status_GVL.strTimeEvent); // RTCManagement

// NETWORK 5
String_Time := CONCAT(STR1 := Status_GVL.strTimeEvent, STR2 := ':');

// NETWORK 6
Status_GVL.Time_PLC := CONCAT(STR1 := String_Time, STR2 := Data_GVL.RTC_DATA.strDT_Second);
END_ACTION

ACTION Test_Outfeed_active:
(**============= Note ================*)
//InputOutput_GVL.TestMode[100] ==> Download Parameter Shuttle Position	
//InputOutput_GVL.TestMode[99]	==> Status Safety
//InputOutput_GVL.TestMode[98]	==> Mute Buzzer
//InputOutput_GVL.TestMode[97]	==> Disable Overflow
//InputOutput_GVL.TestMode[96]	==> Lock Modullar To Run;
//InputOutput_GVL.TestMode[95]	==> Acknowledge Button
//InputOutput_GVL.TestMode[94]	==> Reset Button
//InputOutput_GVL.TestMode[93]	==> Status Running Picking
//InputOutput_GVL.TestMode[92]	==> Bypass Wrapper
//InputOutput_GVL.TestMode[91]	==> Bypass Wrapper Existing


(**============= Test Mode Outfeed ================*)
//=====> Outfeed
InputOutput_GVL.TestMode[1]							:= HMI_GVL.Test_PalletBuffer2_Fwd;
InputOutput_GVL.TestMode[2]							:= HMI_GVL.Test_PalletBuffer1_Fwd;
InputOutput_GVL.TestMode[3]							:= HMI_GVL.Test_PalletOutfeed1_Fwd;
InputOutput_GVL.TestMode[4]							:= HMI_GVL.Test_PalletOutfeed2_Fwd;
InputOutput_GVL.TestMode[5]							:= HMI_GVL.Test_PalletOutfeed3_Fwd;
InputOutput_GVL.TestMode[6]							:= HMI_GVL.Test_PalletOutfeed4_Fwd;
InputOutput_GVL.TestMode[7]							:= HMI_GVL.Test_PalletOutfeed5_Fwd;
InputOutput_GVL.TestMode[8]							:= HMI_GVL.Test_PalletRALifter;
InputOutput_GVL.TestMode[9]							:= HMI_GVL.Test_PalletRATransfer;

IF InputOutput_GVL.Outfeed_stsMachine <> 'Manual' THEN
	HMI_GVL.Test_PalletBuffer2_Fwd					:= FALSE;
	HMI_GVL.Test_PalletBuffer1_Fwd					:= FALSE;
	HMI_GVL.Test_PalletOutfeed1_Fwd					:= FALSE;
	HMI_GVL.Test_PalletOutfeed2_Fwd					:= FALSE;
	HMI_GVL.Test_PalletOutfeed3_Fwd					:= FALSE;
	HMI_GVL.Test_PalletOutfeed4_Fwd					:= FALSE;
	HMI_GVL.Test_PalletOutfeed5_Fwd					:= FALSE;
END_IF

//=====> Shuttle
InputOutput_GVL.TestMode[10]						:= HMI_GVL.Test_ShuttleDrive_Fwd;
InputOutput_GVL.TestMode[11]						:= HMI_GVL.Test_ShuttleDrive_Rev;
InputOutput_GVL.TestMode[12]						:= HMI_GVL.Test_ShuttleLoad_Fwd;
InputOutput_GVL.TestMode[13]						:= HMI_GVL.Test_ShuttleLoad_Rev;
InputOutput_GVL.TestMode[14]						:= HMI_GVL.Test_ShuttleEmpty_Fwd;

IF InputOutput_GVL.Shuttle_stsMachine <> 'Manual' THEN
	HMI_GVL.Test_ShuttleDrive_Fwd					:= FALSE;
	HMI_GVL.Test_ShuttleDrive_Rev					:= FALSE;
	HMI_GVL.Test_ShuttleLoad_Fwd					:= FALSE;
	HMI_GVL.Test_ShuttleLoad_Rev					:= FALSE;
	HMI_GVL.Test_ShuttleEmpty_Fwd					:= FALSE;
END_IF

//=====> Infeed
InputOutput_GVL.TestMode[15]						:= HMI_GVL.Test_BoxInfeed_Fwd;
InputOutput_GVL.TestMode[16]						:= HMI_GVL.Test_BoxStopGo_Fwd;
InputOutput_GVL.TestMode[17]						:= HMI_GVL.Test_BoxBuffer1_Fwd;
InputOutput_GVL.TestMode[18]						:= HMI_GVL.Test_BoxBuffer2_Fwd;
InputOutput_GVL.TestMode[19]						:= HMI_GVL.Test_BoxModullar1_Fwd;
InputOutput_GVL.TestMode[20]						:= HMI_GVL.Test_BoxModullar2_Fwd;
InputOutput_GVL.TestMode[21]						:= HMI_GVL.Test_BoxModullar3_Fwd;
InputOutput_GVL.TestMode[22]						:= HMI_GVL.Test_BoxModullar4_Fwd;
InputOutput_GVL.TestMode[23]						:= HMI_GVL.Test_Stopper1;
InputOutput_GVL.TestMode[24]						:= HMI_GVL.Test_Stopper2;
InputOutput_GVL.TestMode[25]						:= HMI_GVL.Test_Pusher_StopGo_Adv;
InputOutput_GVL.TestMode[26]						:= HMI_GVL.Test_Pusher_StopGo_Rtc;
InputOutput_GVL.TestMode[27]						:= HMI_GVL.Test_Pusher_Buffer1_Adv;
InputOutput_GVL.TestMode[28]						:= HMI_GVL.Test_Pusher_Buffer1_Rtc;
InputOutput_GVL.TestMode[29]						:= HMI_GVL.Test_Pusher_Buffer2_Adv;
InputOutput_GVL.TestMode[30]						:= HMI_GVL.Test_Pusher_Buffer2_Rtc;
InputOutput_GVL.TestMode[31]						:= HMI_GVL.Test_StopperModullar_Adv;
InputOutput_GVL.TestMode[32]						:= HMI_GVL.Test_StopperModullar_Rtc;

IF InputOutput_GVL.Infeed_stsMachine <> 'Manual' THEN
	HMI_GVL.Test_BoxInfeed_Fwd						:= FALSE;
	HMI_GVL.Test_BoxStopGo_Fwd						:= FALSE;
	HMI_GVL.Test_BoxBuffer1_Fwd						:= FALSE;
	HMI_GVL.Test_BoxBuffer2_Fwd						:= FALSE;
	HMI_GVL.Test_BoxModullar1_Fwd					:= FALSE;
	HMI_GVL.Test_BoxModullar2_Fwd					:= FALSE;
	HMI_GVL.Test_BoxModullar3_Fwd					:= FALSE;
	HMI_GVL.Test_BoxModullar4_Fwd					:= FALSE;
	HMI_GVL.Test_Stopper1							:= FALSE;
	HMI_GVL.Test_Stopper2							:= FALSE;
	HMI_GVL.Test_Pusher_StopGo_Adv					:= FALSE;
	HMI_GVL.Test_Pusher_StopGo_Rtc					:= FALSE;
	HMI_GVL.Test_Pusher_Buffer1_Adv					:= FALSE;
	HMI_GVL.Test_Pusher_Buffer1_Rtc					:= FALSE;
	HMI_GVL.Test_Pusher_Buffer2_Adv					:= FALSE;
	HMI_GVL.Test_Pusher_Buffer2_Rtc					:= FALSE;
END_IF
END_ACTION

END_PROGRAM

(* stored: Version 1.1.0.1, ProductVersion 3.1.4024.12
   POU Backbone: Id {5d8e9ef5-a3d3-4130-8f7b-0d6c323cc7fd}, SpecialFunc None
   Action Error_Outfeed_active: Id {c0d15e54-5ad9-4f3f-81db-6be6aa6117b0}
   Action FGHS_DataCollect_active: Id {77a263b6-5ae2-4bbb-9273-00ed46aba089}
   Action FGHS_DataTraffict_active: Id {cda21a1b-26f0-4096-a9f2-22d3c98dc177}
   Action Indicator_active: Id {094d60b3-0420-4a73-b74d-3600408507ff}
   Action OEE_active: Id {e5065722-83c5-4fbb-bec6-9e88f3fc3002}
   Action Parameter_Outfeed_active: Id {bfa80fdd-0716-44d0-a965-1973c10453bd}
   Action Recipe_active: Id {272f3086-172f-436f-8fca-e3aa00ca9f0f}
   Action RTC_Management_active: Id {e3c35964-3d93-4d5f-afd5-bb34df6fe18f}
   Action Test_Outfeed_active: Id {89aac1cc-1fd1-49bd-83ed-18976c5df5c2} *)
